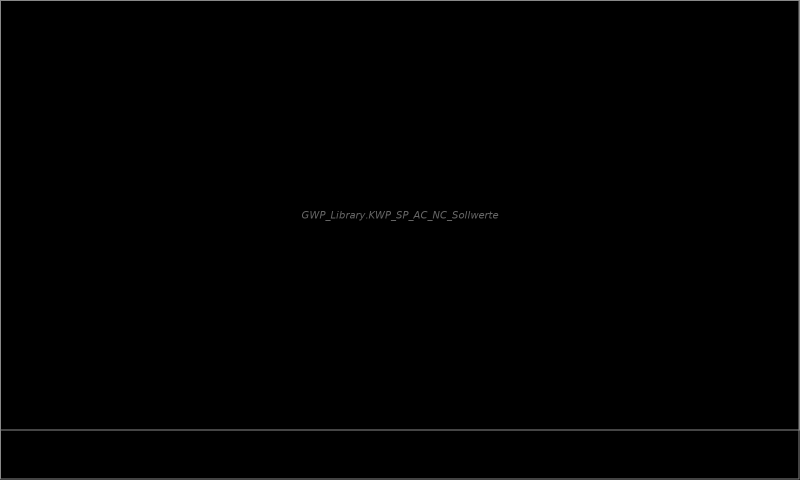
VISUALIZATION KWP_SP_AC_NC_Sollwerte  // 800x480
    Frame (0,0 800x430)
        shows GWP_Library.KWP_SP_AC_NC_Sollwerte(FB_KWP_SP_AC_NC := Main.KWP_SP_AC_NC_0, FB_Kreis_3KO := Main.Kreis_3KO_0, FB_VD := Main.VD_0, FB_Init_1 := Main.Init_0)
END_VISUALIZATION

(* stored: Version 1.1.0.1, ProductVersion 3.1.4022.6
   Visu KWP_SP_AC_NC_Sollwerte: Id {023b4151-041f-4ddd-a28e-d6790db058dd} *)
